FUNCTION_BLOCK CL_AxisDriverL1LeftBack EXTENDS CL_AxisDriverAX8206
VAR
END_VAR

SUPER^();

METHOD PROTECTED InitDefect : BOOL
VAR_INPUT
END_VAR
InitDefect := true;
END_METHOD

END_FUNCTION_BLOCK

(* stored: Version 1.1.0.1, ProductVersion 3.1.4024.12
   POU CL_AxisDriverL1LeftBack: Id {fa1ea31c-ec11-4e67-b56f-8859648caf74}, SpecialFunc None
   Method InitDefect: Id {1becdde8-68ff-49f8-a75c-c8d1d6094ec3} *)
